PROGRAM MAIN
VAR
END_VAR

PLC_PRG();

END_PROGRAM

(* stored: Version 1.1.0.1, ProductVersion 3.1.4022.12
   POU MAIN: Id {b0c72497-773d-4397-b6c2-cabc9094ffb5}, SpecialFunc None *)
